FUNCTION_BLOCK ADD_UINT (* IEC 61131-3 UINT Addition *)
  (* Standard: 61131-3 *)
  (* Version 0.0, 2006-09-11, JHC, Holobloc Inc *)
  (* Compiler header: package fb.rt.plc.math; *)
  (* Compiler classdef: (Math.min(65535, IN1 + IN2 )) *)
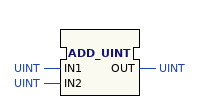
  VAR_INPUT
    IN1 : UINT; (* Augend *)
    IN2 : UINT; (* Addend *)
  END_VAR
  VAR_OUTPUT
    OUT : UINT; (* Sum *)
  END_VAR
END_FUNCTION_BLOCK
